# EPICS StreamDevice protocol: devJDQ016.proto
InTerminator = "";
OutTerminator = "";
setRelay0 {
    out "\xCC\xDD\xA1\x01%{\x00\x00\x00\x01|\x00\x01\x00\x01}%2<sum>%2<sum>";
    in "%s";
}
setRelay1 {
    out "\xCC\xDD\xA1\x01%{\x00\x00\x00\x02|\x00\x02\x00\x02}%2<sum>%2<sum>";
    in "%s";
}

setRelay2 {
    out "\xCC\xDD\xA1\x01%{\x00\x00\x00\x04|\x00\x04\x00\x04}%2<sum>%2<sum>";
    in "%s";
}

setRelay3 {
    out "\xCC\xDD\xA1\x01%{\x00\x00\x00\x08|\x00\x08\x00\x08}%2<sum>%2<sum>";
    in "%s";
}

setRelay4 {
    out "\xCC\xDD\xA1\x01%{\x00\x00\x00\x10|\x00\x10\x00\x10}%2<sum>%2<sum>";
    in "%s";
}

setRelay5 {
    out "\xCC\xDD\xA1\x01%{\x00\x00\x00\x20|\x00\x20\x00\x20}%2<sum>%2<sum>";
    in "%s";
}

setRelay6 {
    out "\xCC\xDD\xA1\x01%{\x00\x00\x00\x40|\x00\x40\x00\x40}%2<sum>%2<sum>";
    in "%s";
}

setRelay7 {
    out "\xCC\xDD\xA1\x01%{\x00\x00\x00\x80|\x00\x80\x00\x80}%2<sum>%2<sum>";
    in "%s";
}

setRelay8 {
    out "\xCC\xDD\xA1\x01%{\x00\x00\x01\x00|\x01\x00\x01\x00}%2<sum>%2<sum>";
    in "%s";
}

setRelay9 {
    out "\xCC\xDD\xA1\x01%{\x00\x00\x02\x00|\x02\x00\x02\x00}%2<sum>%2<sum>";
    in "%s";
}

setRelayA {
    out "\xCC\xDD\xA1\x01%{\x00\x00\x04\x00|\x04\x00\x04\x00}%2<sum>%2<sum>";
    in "%s";
}

setRelayB {
    out "\xCC\xDD\xA1\x01%{\x00\x00\x08\x00|\x08\x00\x08\x00}%2<sum>%2<sum>";
    in "%s";
}

setRelayC {
    out "\xCC\xDD\xA1\x01%{\x00\x00\x10\x00|\x10\x00\x10\x00}%2<sum>%2<sum>";
    in "%s";
}

setRelayD {
    out "\xCC\xDD\xA1\x01%{\x00\x00\x20\x00|\x20\x00\x20\x00}%2<sum>%2<sum>";
    in "%s";
}

setRelayE {
    out "\xCC\xDD\xA1\x01%{\x00\x00\x40\x00|\x40\x00\x40\x00}%2<sum>%2<sum>";
    in "%s";
}

setRelayF {
    out "\xCC\xDD\xA1\x01%{\x00\x00\x80\x00|\x80\x00\x80\x00}%2<sum>%2<sum>";
    in "%s";
}

set {
    out "\xCC\xDD\xA1\x01\$1%2<sum>%2<sum>";
    in "%s";
}

setAll {
    out "\xCC\xDD\xA1\x01%{\x00\x00\xFF\xFF|\xFF\xFF\xFF\xFF}%2<sum>%2<sum>";
    in "%s";
}

readRelayState {
	wait 50;
	out "\xCC\xDD\xB0\x01\x00\x00\x0D\xBE\x7C";
	in "%*4c%2r[^\x0D]";
#	in "\xAA\xBB\xB0\x01%2r\x0D%2<sum>%2<sum>";
}

readInState {
	wait 50;
	out "\xCC\xDD\xC0\x01\x00\x00\x0D\xCE\x9C";
#	in "\xAA\xBB\xC0\x01%2x\x0D%2<sum>%2<sum>";
	in "%*4c%2r[^\x0D]";
}
